// TIA Portal V19 export
TYPE "Positioning_DOL_Machine_DataIn"
// stored: Access Published
   STRUCT
      PB : "Ax_PB";
      LS_Minus : Bool;
      LS_Plus : Bool;
      Fan_M_ThermalProtection : Bool := FALSE;
      Fan_M_Feedback : Bool;
      Brake_M_Q : Bool;   // SINAMICS is controlling the Brake Opening
      Brake_M_Feedback : Bool := TRUE;   // If brake not available leave this value at TRUE
   END_STRUCT;
END_TYPE
